{attribute addProperty BoxType "IL2300-B110-0017"}
{attribute addProperty Id "Term_20KL_5BCCED4C00Term_391_Ix1000KL_9BB4615400"}
{attribute addProperty CRC "1547459922"}
{attribute addProperty SizeInBites "0"}
{attribute addProperty SizeInBytes "0"}
TYPE A_0020_IL2300_B110_0017_5C3C5D52 EXTENDS IL2300_4487A81F :
STRUCT
	{attribute addProperty Name "Term_20"}
	Term_20 : KL_5BCCED4C;
	{attribute addProperty Name "Term_391_Ix1000"}
	Term_391_Ix1000 : KL_9BB46154;
END_STRUCT
END_TYPE

(* stored: Version 1.2.0.0, ProductVersion 3.1.4024.9
   DUT A_0020_IL2300_B110_0017_5C3C5D52: Id {f7974a33-88b5-44a7-9f21-6e56ba4be0ab} *)
